FUNCTION_BLOCK Physical_Plant_Simulation (* Composite Function Block Type *)
  (* Standard: 61499-2 *)
  (* Version 0.0, 12/12/2023, Cheyan, Schneider Electric, template *)
  PACKAGE Main;
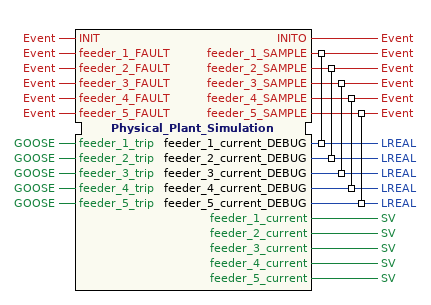
  EVENT_INPUT
    INIT; (* Initialization Request *)
    feeder_1_FAULT;
    feeder_2_FAULT;
    feeder_3_FAULT;
    feeder_4_FAULT;
    feeder_5_FAULT;
  END_EVENT
  EVENT_OUTPUT
    INITO; (* Initialization Confirm *)
    feeder_1_SAMPLE WITH feeder_1_current_DEBUG;
    feeder_2_SAMPLE WITH feeder_2_current_DEBUG;
    feeder_3_SAMPLE WITH feeder_3_current_DEBUG;
    feeder_4_SAMPLE WITH feeder_4_current_DEBUG;
    feeder_5_SAMPLE WITH feeder_5_current_DEBUG;
  END_EVENT
  VAR_OUTPUT
    feeder_1_current_DEBUG : LREAL; (* Output event qualifier *)
    feeder_2_current_DEBUG : LREAL; (* Output event qualifier *)
    feeder_3_current_DEBUG : LREAL; (* Output event qualifier *)
    feeder_4_current_DEBUG : LREAL; (* Output event qualifier *)
    feeder_5_current_DEBUG : LREAL; (* Output event qualifier *)
  END_VAR
  SOCKETS
    feeder_1_trip : GOOSE;
    feeder_2_trip : GOOSE;
    feeder_3_trip : GOOSE;
    feeder_4_trip : GOOSE;
    feeder_5_trip : GOOSE;
  END_SOCKETS
  PLUGS
    feeder_1_current : SV;
    feeder_2_current : SV;
    feeder_3_current : SV;
    feeder_4_current : SV;
    feeder_5_current : SV;
  END_PLUGS
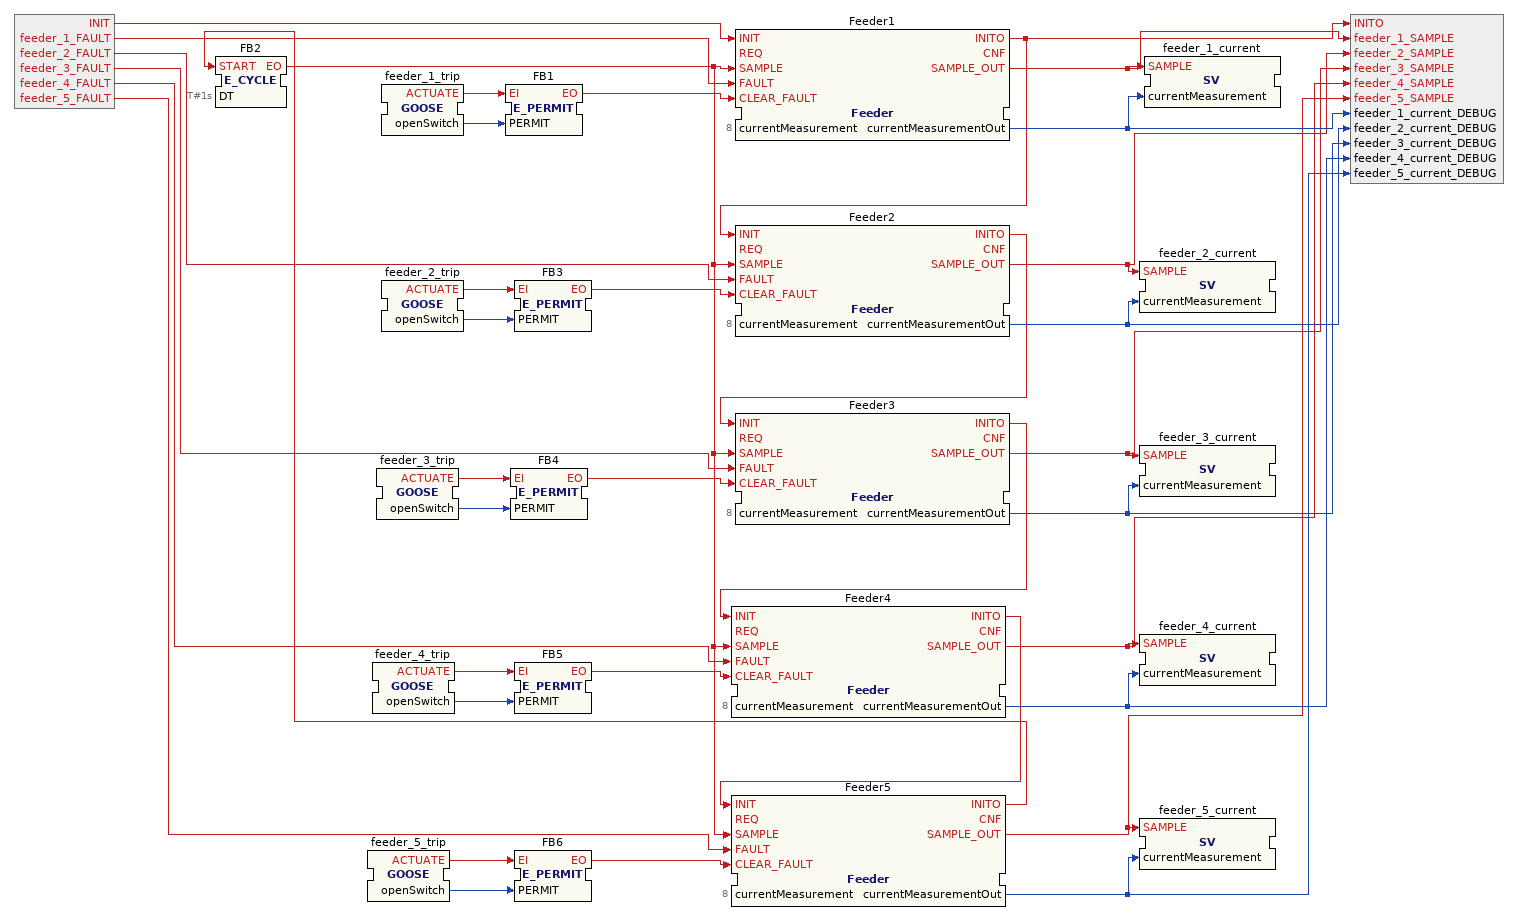
  FBS
    Feeder1 : Feeder(currentMeasurement := 8);
    FB2 : E_CYCLE(DT := T#1s);
    Feeder2 : Feeder(currentMeasurement := 8);
    Feeder3 : Feeder(currentMeasurement := 8);
    Feeder4 : Feeder(currentMeasurement := 8);
    Feeder5 : Feeder(currentMeasurement := 8);
    FB1 : E_PERMIT;
    FB3 : E_PERMIT;
    FB4 : E_PERMIT;
    FB5 : E_PERMIT;
    FB6 : E_PERMIT;
  END_FBS
  EVENT_CONNECTIONS
    FB2.EO TO Feeder1.SAMPLE;
    INIT TO Feeder1.INIT;
    Feeder1.INITO TO Feeder2.INIT;
    Feeder2.INITO TO Feeder3.INIT;
    Feeder3.INITO TO Feeder4.INIT;
    Feeder4.INITO TO Feeder5.INIT;
    Feeder5.INITO TO FB2.START;
    feeder_1_FAULT TO Feeder1.FAULT;
    feeder_2_FAULT TO Feeder2.FAULT;
    FB2.EO TO Feeder2.SAMPLE;
    FB2.EO TO Feeder3.SAMPLE;
    feeder_3_FAULT TO Feeder3.FAULT;
    feeder_4_FAULT TO Feeder4.FAULT;
    FB2.EO TO Feeder4.SAMPLE;
    FB2.EO TO Feeder5.SAMPLE;
    feeder_5_FAULT TO Feeder5.FAULT;
    Feeder1.SAMPLE_OUT TO feeder_1_SAMPLE;
    Feeder1.INITO TO INITO;
    Feeder2.SAMPLE_OUT TO feeder_2_SAMPLE;
    Feeder3.SAMPLE_OUT TO feeder_3_SAMPLE;
    Feeder4.SAMPLE_OUT TO feeder_4_SAMPLE;
    Feeder5.SAMPLE_OUT TO feeder_5_SAMPLE;
    Feeder1.SAMPLE_OUT TO feeder_1_current.SAMPLE;
    Feeder2.SAMPLE_OUT TO feeder_2_current.SAMPLE;
    Feeder3.SAMPLE_OUT TO feeder_3_current.SAMPLE;
    Feeder4.SAMPLE_OUT TO feeder_4_current.SAMPLE;
    Feeder5.SAMPLE_OUT TO feeder_5_current.SAMPLE;
    feeder_1_trip.ACTUATE TO FB1.EI;
    FB1.EO TO Feeder1.CLEAR_FAULT;
    feeder_2_trip.ACTUATE TO FB3.EI;
    FB3.EO TO Feeder2.CLEAR_FAULT;
    feeder_3_trip.ACTUATE TO FB4.EI;
    FB4.EO TO Feeder3.CLEAR_FAULT;
    feeder_4_trip.ACTUATE TO FB5.EI;
    FB5.EO TO Feeder4.CLEAR_FAULT;
    feeder_5_trip.ACTUATE TO FB6.EI;
    FB6.EO TO Feeder5.CLEAR_FAULT;
  END_CONNECTIONS
  DATA_CONNECTIONS
    Feeder1.currentMeasurementOut TO feeder_1_current_DEBUG;
    Feeder2.currentMeasurementOut TO feeder_2_current_DEBUG;
    Feeder3.currentMeasurementOut TO feeder_3_current_DEBUG;
    Feeder4.currentMeasurementOut TO feeder_4_current_DEBUG;
    Feeder5.currentMeasurementOut TO feeder_5_current_DEBUG;
    Feeder1.currentMeasurementOut TO feeder_1_current.currentMeasurement;
    Feeder2.currentMeasurementOut TO feeder_2_current.currentMeasurement;
    Feeder3.currentMeasurementOut TO feeder_3_current.currentMeasurement;
    Feeder4.currentMeasurementOut TO feeder_4_current.currentMeasurement;
    Feeder5.currentMeasurementOut TO feeder_5_current.currentMeasurement;
    feeder_1_trip.openSwitch TO FB1.PERMIT;
    feeder_2_trip.openSwitch TO FB3.PERMIT;
    feeder_3_trip.openSwitch TO FB4.PERMIT;
    feeder_4_trip.openSwitch TO FB5.PERMIT;
    feeder_5_trip.openSwitch TO FB6.PERMIT;
  END_CONNECTIONS
END_FUNCTION_BLOCK
